TYPE (* IEC61131-3, Table 14#5 *)
  (* Standard: 1131-3 *)
  (* Version 0.0, 1/8/2024, Cheyan, Schneider Electric, Template *)
  PACKAGE Main;
  {SET_ATTRIBUTE(nxtDataType, UylDVgj4yyFp3fGyCOavW/kuNztsjOZEwZQ9Ck6MPeX3f9a09pxMlQ19d25XPF9/BgRd1+6DF/gocA8GhVf07AifoybxmGDkJ2qqfcE/unnJds7ZkdI9kg==)}
  SPC_CTLMODEL : STRUCT
    ctlModel : CtlModels;
  END_STRUCT;
END_TYPE
